// One row returned by a SELECT from the ds table
TYPE ST_DbRecord : STRUCT
  id        : DINT;
  timestamp : DT;
  value     : REAL;
END_STRUCT
END_TYPE

(* stored: Version 1.1.0.1, ProductVersion 3.1.4026.18
   DUT ST_DbRecord: Id {681761f0-f6a6-436d-95f0-ee77c76f00f0} *)
